// Mitsubishi GX Works2 project: SEQUENCE_TIMER2   PLC: Q03UDV

PROGRAM MAIN
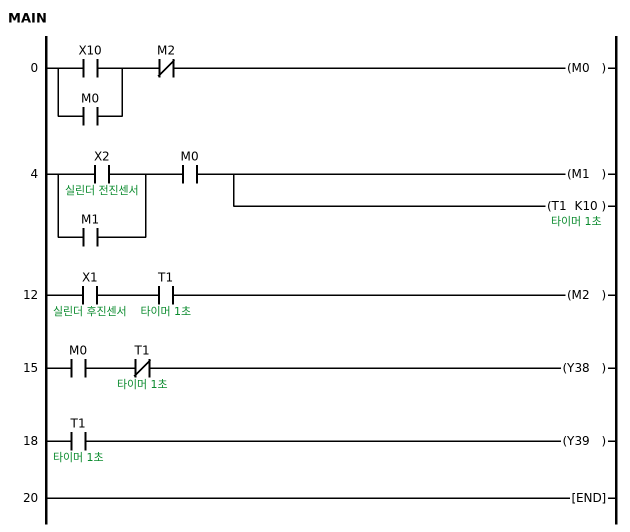
0     LD      X10
      OR      M0
      ANI     M2
      OUT     M0
4     LD      X2  ; 실린더 전진센서
      OR      M1
      AND     M0
      OUT     M1
      OUT     T1 K10  ; 타이머 1초
12    LD      X1  ; 실린더 후진센서
      AND     T1  ; 타이머 1초
      OUT     M2
15    LD      M0
      ANI     T1  ; 타이머 1초
      OUT     Y38
18    LD      T1  ; 타이머 1초
      OUT     Y39
20    END
END_PROGRAM
